TYPE ST_AxisIN :
STRUCT
	

bPower			:	BOOL;
nOverride		:	INT;

bAbs			:	BOOL;
fVelocity		:	LREAL;
fPos			:	LREAL;
            	
bCamIN			:	BOOL;
nCamTableID		:	UDINT;
bCamOUT			:	BOOL;
            	
bStop			:	BOOL;
            	
bReset			:	BOOL;
            	
bRead			:	BOOL;
            	
bWrite			:	BOOL;
nCamTableIdWr	:	UDINT;

END_STRUCT
END_TYPE

(* stored: Version 1.1.0.1, ProductVersion 3.1.4022.18
   DUT ST_AxisIN: Id {6aea9bc0-1f3b-4bca-b199-c2089a07b8f2} *)
